# EPICS StreamDevice protocol: k2000/proto/k2000.proto
Terminator = CR LF;

read {
	out "READ?";
	in "%f";
}
